{attribute 'qualified_only'}
{attribute 'strict'}
{attribute 'to_string'}
TYPE e_db_steel_status :
(
	inSide := 1, // 入料  
	holding := 2, // 暫存中(在吊掛區等待進入料架)
	waitLoading := 3, // 等待上料(在料架上等待，後進入機台)
	alignment := 10, // 無靠邊插單
	inserts := 11, // 插單
	machining := 20, // 加工中
	waitUnloading := 30, // 等待下料(在料架上等待，後進入出料吊掛區或其他機台)
	finish := 40, //加工完成
	paired := 100, // 已配對
	pairing := 101, // 配對中
	waitPaired := 102, // 等待配對
	pairedCancel := 108, // 配對取消
	pairedFailed := 109, // 配對失敗
	dxfTransferring := 996, // DXF 傳輸中
	connectedFailed := 997, // 連線失敗
	transformFailed := 998, // 轉換失敗
	unknown := 999 // 未知
);
END_TYPE
//  unknown = '999 '

(* stored: Version 1.1.0.1, ProductVersion 3.1.4026.13
   EnumerationTextList e_db_steel_status: Id {305133de-f98a-44a9-a26a-0fb90dd07f0e} *)
